(* PLC project plc_garden_controller2.project, CODESYS CODESYS V3.5 SP16 *)
(* stored: creationDateTime 2021-03-27T17:20:38.1897763, modificationDateTime 2021-03-27T17:20:27.5902223 *)

TYPE Flower_typ : STRUCT
  x : INT;
  y : INT;
  alpha : BYTE := 255;  (* Alpha channel *)
  red : BYTE := 2;  (* Red color channel *)
  green : BYTE := 253;  (* Green color channel *)
  blue : BYTE := 0;  (* Blue color channel *)
  color : DWORD;  (* Color variable to be used in the graphics *)
  hum : REAL := 100;
END_STRUCT;
END_TYPE

PROGRAM simu
  VAR
    clock : ClockPulse;  (* Clock pulse for the program *)
    i : UINT;
    vTest : BOOL;
    vGarden1 : ARRAY[0..24] OF Flower_typ;
    vGarden2 : ARRAY[0..24] OF Flower_typ;
    vGarden3 : ARRAY[0..24] OF Flower_typ;
    vGarden4 : ARRAY[0..24] OF Flower_typ;
  END_VAR

                    clock(f:=T#0.01S);

(*Run the garden simulators*)
garden1();
garden2();
garden3();
garden4();
                  

ACTION garden1:
                        (*COLOR : 16# XX XX XX XX*)
(*            A  R  G  B *)
FOR i:=0 TO 24 DO
	(*Simulate the humidity of one flower cell*)
	(*If not being watered, it slowly looses humidity*)
	vGarden1[i].hum := MAX(0, vGarden1[i].hum - 0.5 * BOOL_TO_REAL(clock.pulse));
	
	(*If the watering platform is above the cell, water valve is open and tank has water, increase the humidity*)
	IF vTest THEN
		vGarden1[i].hum := vGarden1[i].hum + 2 * BOOL_TO_REAL(clock.pulse);
	END_IF
	
	(*Simulate flowers response to the humidity of the cell*)
	IF vGarden1[i].hum <= 0 OR vGarden1[i].hum >= 200 THEN
		(*Flower starts decaying if not enough or too much humiditiy*)
		(*Change color towards red*)
		vGarden1[i].red := vGarden1[i].red + 1 * BOOL_TO_BYTE(clock.pulse);
		vGarden1[i].green := vGarden1[i].green - 1 * BOOL_TO_BYTE(clock.pulse AND vGarden1[i].red > 253);
	ELSE
		IF vGarden1[i].red < 200 AND vGarden1[i].green > 1 THEN
			(*Flower gets better much faster than it dies*)
			(*Change color towards green*)
			vGarden1[i].green := vGarden1[i].green + 1 * BOOL_TO_BYTE(clock.pulse);
			vGarden1[i].red := vGarden1[i].red - 1 * BOOL_TO_BYTE(clock.pulse AND vGarden1[i].green > 253);
		(*ELSE It is dead for good*)
		END_IF
	END_IF
	vGarden1[i].red := LIMIT(1, vGarden1[i].red, 254);
	vGarden1[i].green := LIMIT(1, vGarden1[i].green, 254);
	
	(*Combine the channel bytes into dword color*)
	vGarden1[i].color := BYTES_TO_DWORD(B0 := vGarden1[i].blue,B1 := vGarden1[i].green,
										B2 := vGarden1[i].red, B3 := vGarden1[i].alpha);
END_FOR
                      
END_ACTION

ACTION garden2:
                        (*COLOR : 16# XX XX XX XX*)
(*            A  R  G  B *)
FOR i:=0 TO 24 DO
	(*Simulate the humidity of one flower cell*)
	(*If not being watered, it slowly looses humidity*)
	vGarden2[i].hum := MAX(0, vGarden2[i].hum - 0.5 * BOOL_TO_REAL(clock.pulse));
	
	(*If the watering platform is above the cell, water valve is open and tank has water, increase the humidity*)
	IF vTest THEN
		vGarden2[i].hum := vGarden2[i].hum + 2 * BOOL_TO_REAL(clock.pulse);
	END_IF
	
	(*Simulate flowers response to the humidity of the cell*)
	IF vGarden2[i].hum <= 0 OR vGarden2[i].hum >= 200 THEN
		(*Flower starts decaying if not enough or too much humiditiy*)
		(*Change color towards red*)
		vGarden2[i].red := vGarden2[i].red + 1 * BOOL_TO_BYTE(clock.pulse);
		vGarden2[i].green := vGarden2[i].green - 1 * BOOL_TO_BYTE(clock.pulse AND vGarden2[i].red > 253);
	ELSE
		IF vGarden2[i].red < 200 AND vGarden2[i].green > 1 THEN
			(*Flower gets better much faster than it dies*)
			(*Change color towards green*)
			vGarden2[i].green := vGarden2[i].green + 1 * BOOL_TO_BYTE(clock.pulse);
			vGarden2[i].red := vGarden2[i].red - 1 * BOOL_TO_BYTE(clock.pulse AND vGarden2[i].green > 253);
		(*ELSE It is dead for good*)
		END_IF
	END_IF
	vGarden2[i].red := LIMIT(1, vGarden2[i].red, 254);
	vGarden2[i].green := LIMIT(1, vGarden2[i].green, 254);
	
	(*Combine the channel bytes into dword color*)
	vGarden2[i].color := BYTES_TO_DWORD(B0 := vGarden2[i].blue,B1 := vGarden2[i].green,
										B2 := vGarden2[i].red, B3 := vGarden2[i].alpha);
END_FOR
                      
END_ACTION

ACTION garden3:
                        (*COLOR : 16# XX XX XX XX*)
(*            A  R  G  B *)
FOR i:=0 TO 24 DO
	(*Simulate the humidity of one flower cell*)
	(*If not being watered, it slowly looses humidity*)
	vGarden3[i].hum := MAX(0, vGarden3[i].hum - 0.5 * BOOL_TO_REAL(clock.pulse));
	
	(*If the watering platform is above the cell, water valve is open and tank has water, increase the humidity*)
	IF vTest THEN
		vGarden3[i].hum := vGarden3[i].hum + 2 * BOOL_TO_REAL(clock.pulse);
	END_IF
	
	(*Simulate flowers response to the humidity of the cell*)
	IF vGarden3[i].hum <= 0 OR vGarden3[i].hum >= 200 THEN
		(*Flower starts decaying if not enough or too much humiditiy*)
		(*Change color towards red*)
		vGarden3[i].red := vGarden3[i].red + 1 * BOOL_TO_BYTE(clock.pulse);
		vGarden3[i].green := vGarden3[i].green - 1 * BOOL_TO_BYTE(clock.pulse AND vGarden3[i].red > 253);
	ELSE
		IF vGarden3[i].red < 200 AND vGarden3[i].green > 1 THEN
			(*Flower gets better much faster than it dies*)
			(*Change color towards green*)
			vGarden3[i].green := vGarden3[i].green + 1 * BOOL_TO_BYTE(clock.pulse);
			vGarden3[i].red := vGarden3[i].red - 1 * BOOL_TO_BYTE(clock.pulse AND vGarden3[i].green > 253);
		(*ELSE It is dead for good*)
		END_IF
	END_IF
	vGarden3[i].red := LIMIT(1, vGarden3[i].red, 254);
	vGarden3[i].green := LIMIT(1, vGarden3[i].green, 254);
	
	(*Combine the channel bytes into dword color*)
	vGarden3[i].color := BYTES_TO_DWORD(B0 := vGarden3[i].blue,B1 := vGarden3[i].green,
										B2 := vGarden3[i].red, B3 := vGarden3[i].alpha);
END_FOR
                      
END_ACTION

ACTION garden4:
                        (*COLOR : 16# XX XX XX XX*)
(*            A  R  G  B *)
FOR i:=0 TO 24 DO
	(*Simulate the humidity of one flower cell*)
	(*If not being watered, it slowly looses humidity*)
	vGarden4[i].hum := MAX(0, vGarden4[i].hum - 0.5 * BOOL_TO_REAL(clock.pulse));
	
	(*If the watering platform is above the cell, water valve is open and tank has water, increase the humidity*)
	IF vTest THEN
		vGarden4[i].hum := vGarden4[i].hum + 2 * BOOL_TO_REAL(clock.pulse);
	END_IF
	
	(*Simulate flowers response to the humidity of the cell*)
	IF vGarden4[i].hum <= 0 OR vGarden4[i].hum >= 200 THEN
		(*Flower starts decaying if not enough or too much humiditiy*)
		(*Change color towards red*)
		vGarden4[i].red := vGarden4[i].red + 1 * BOOL_TO_BYTE(clock.pulse);
		vGarden4[i].green := vGarden4[i].green - 1 * BOOL_TO_BYTE(clock.pulse AND vGarden4[i].red > 253);
	ELSE
		IF vGarden4[i].red < 200 AND vGarden4[i].green > 1 THEN
			(*Flower gets better much faster than it dies*)
			(*Change color towards green*)
			vGarden4[i].green := vGarden4[i].green + 1 * BOOL_TO_BYTE(clock.pulse);
			vGarden4[i].red := vGarden4[i].red - 1 * BOOL_TO_BYTE(clock.pulse AND vGarden4[i].green > 253);
		(*ELSE It is dead for good*)
		END_IF
	END_IF
	vGarden4[i].red := LIMIT(1, vGarden4[i].red, 254);
	vGarden4[i].green := LIMIT(1, vGarden4[i].green, 254);
	
	(*Combine the channel bytes into dword color*)
	vGarden4[i].color := BYTES_TO_DWORD(B0 := vGarden4[i].blue,B1 := vGarden4[i].green,
										B2 := vGarden4[i].red, B3 := vGarden4[i].alpha);
END_FOR
                      
END_ACTION
END_PROGRAM

FUNCTION BYTES_TO_DWORD : DWORD
  VAR_INPUT
    B0 : BYTE;  (* Least significant byte *)
    B1 : BYTE;  (* Byte two *)
    B2 : BYTE;  (* Byte three *)
    B3 : BYTE;  (* Highest significant byte *)
  END_VAR

                    BYTES_TO_DWORD.0 := B0.0;
BYTES_TO_DWORD.1 := B0.1;
BYTES_TO_DWORD.2 := B0.2;
BYTES_TO_DWORD.3 := B0.3;
BYTES_TO_DWORD.4 := B0.4;
BYTES_TO_DWORD.5 := B0.5;
BYTES_TO_DWORD.6 := B0.6;
BYTES_TO_DWORD.7 := B0.7;

BYTES_TO_DWORD.8 := B1.0;
BYTES_TO_DWORD.9 := B1.1;
BYTES_TO_DWORD.10 := B1.2;
BYTES_TO_DWORD.11 := B1.3;
BYTES_TO_DWORD.12 := B1.4;
BYTES_TO_DWORD.13 := B1.5;
BYTES_TO_DWORD.14 := B1.6;
BYTES_TO_DWORD.15 := B1.7;

BYTES_TO_DWORD.16 := B2.0;
BYTES_TO_DWORD.17 := B2.1;
BYTES_TO_DWORD.18 := B2.2;
BYTES_TO_DWORD.19 := B2.3;
BYTES_TO_DWORD.20 := B2.4;
BYTES_TO_DWORD.21 := B2.5;
BYTES_TO_DWORD.22 := B2.6;
BYTES_TO_DWORD.23 := B2.7;

BYTES_TO_DWORD.24 := B3.0;
BYTES_TO_DWORD.25 := B3.1;
BYTES_TO_DWORD.26 := B3.2;
BYTES_TO_DWORD.27 := B3.3;
BYTES_TO_DWORD.28 := B3.4;
BYTES_TO_DWORD.29 := B3.5;
BYTES_TO_DWORD.30 := B3.6;
BYTES_TO_DWORD.31 := B3.7;
RETURN;
                  
END_FUNCTION

FUNCTION_BLOCK ClockPulse
  VAR_INPUT
    f : TIME := TIME#500ms;  (* Oscillate once per f *)
  END_VAR
  VAR_OUTPUT
    pulse : BOOL;  (* Pulse for use. One cycle *)
  END_VAR
  VAR
    edge : R_TRIG;
    clock : BLINK;
  END_VAR

                    clock(ENABLE:=TRUE, TIMELOW:=f, TIMEHIGH:=f);
edge(CLK:=clock.OUT);
pulse := edge.Q;
                  
END_FUNCTION_BLOCK

CONFIGURATION SoftPLC
  RESOURCE Application ON PLC
    TASK VISU_TASK(INTERVAL := T#100ms, PRIORITY := 31);
    TASK Task(INTERVAL := T#20ms, PRIORITY := 1);
    PROGRAM VisuElems.Visu_Prg WITH VISU_TASK : VisuElems.Visu_Prg;
    PROGRAM simu WITH Task : simu;
  END_RESOURCE
END_CONFIGURATION
